FUNCTION_BLOCK Infeed EXTENDS FB_PackML_BaseModule
VAR
END_VAR

END_FUNCTION_BLOCK

(* stored: Version 1.1.0.1
   POU Infeed: Id {4745b5cb-9cfa-45ed-bd8a-2d7985365640}, SpecialFunc None *)
